// TIA Portal V16 export
// export: Created 2021-11-12T13:33:06.5426494Z, ExportSetting WithDefaults, DisplayName Totally Integrated Automation Portal, DisplayVersion V16 Update 3, DisplayName TIA Portal Version Control Interface, DisplayVersion V16 Update 2, DisplayName TIA Portal Openness, DisplayVersion V16 Update 3, DisplayName SINAMICS Startdrive Advanced, DisplayVersion V16 Update 5, DisplayName SINAMICS Startdrive G130, G150, S120, S150, SINAMICS MV, S210, DisplayVersion V16 Update 5, DisplayName SINAMICS Startdrive G110M, G120, G120C, G120D, G120P, G115D, DisplayVersion V16 Update 5, DisplayName STEP 7 Professional, DisplayVersion V16 Update 3, DisplayName STEP 7 Safety, DisplayVersion V16, DisplayName WinCC UA Professional, DisplayVersion V16 Update 3
FUNCTION_BLOCK "Station410"   // FB83, LAD
{ S7_Optimized_Access := 'TRUE' }
VERSION : 0.1
// stored: AutoNumber true, IsIECCheckEnabled false, IsRetainMemResEnabled false, MemoryReserve 100, SetENOAutomatically false, UDAEnableTagReadback false
   VAR
      "SF_EQ01-MA01" : "STD_Drive1";   // Water pump (P31)
      "SF_EQ01-MA02" : "STD_Valve2WB";   // Valve with servomotor (A1417)
      "SF_EQ01-MA03" : "STD_Valve2WB";   // Valve with servomotor (A1414)
      "SF_EQ01-MA04" : "STD_Valve2WB";   // Valve with servomotor (A1411)
      "SF_UC11-TA01" { S7_SetPoint := 'True'} : "STD_Siemens_G120_CU240E_2_PN";   // Conveyor
      SF_Alarm1 { S7_SetPoint := 'True'} : "STD_DI_Mon";   // Sensor Max level active and sensor Min level
      SF_Alarm2 { S7_SetPoint := 'True'} : "STD_DI_Mon";   // Sensor Min level active and analog level sensor under 10%
      SF_Alarm3 { S7_SetPoint := 'True'} : "STD_DI_Mon";   // Analog level sensor over 40% and sensor min level not active
      SF_Alarm4 { S7_SetPoint := 'True'} : "STD_DI_Mon";   // Water temperature high
      SF_Alarm5 { S7_SetPoint := 'True'} : "STD_DI_Mon";   // Water temperature low
      SF_Alarm6 { S7_SetPoint := 'True'} : "STD_DI_Mon";   // Water level high
      SF_Alarm7 { S7_SetPoint := 'True'} : "STD_DI_Mon";   // BSN 5 tacts and water level NOK
      SF_Alarm8 { S7_SetPoint := 'True'} : "STD_DI_Mon";   // Filling and no water level change
      SF_Alarm9 { S7_SetPoint := 'True'} : "STD_DI_Mon";   // Drain and no water level change
      SS_Cooling : Struct
         LiqTemp : Real;   // Real temperature of liquid
         HystMin : Real;   // Minimal hysteresis of requested temperature for cooling liquid
         HystMax : Real;   // Maximal hysteresis of requested temperature for cooling liquid
         RunPump : Bool;
         RegEn : Bool;   // Enable regulation
      END_STRUCT;
      SR_TmpWaterLevel : Real;
      SB1_PowerOk { S7_SetPoint := 'True'} : Bool;
      SF_TimerWaterHom { S7_SetPoint := 'True'} : TON_TIME;
   END_VAR
   VAR_TEMP
      TS_EQ01MA01 : "UDT_DriveControl";   // Water pump (P31)
      TS_EQ01MA02 : "UDT_DriveControl";   // Valve with servomotor (A1417)
      TS_EQ01MA03 : "UDT_DriveControl";   // Valve with servomotor (A1414)
      TS_EQ01MA04 : "UDT_DriveControl";   // Valve with servomotor (A1411)
      TS_UC11TA01 : Struct   // Conveyor
         ReqDir1 : Bool;   // Move in direction 1
         ReqDir2 : Bool;   // Move in direction 2
         AckErr : Bool;   // Acknowledge error
         SpeedSP : Real;   // Speed setpoint
      END_STRUCT;
      TS_CirculationValve : Struct
         HystMin : Real;
         HystMax : Real;
         SP : Real;
      END_STRUCT;
      TB1_WaterHom : Bool;   // Water homogenization is not done
   END_VAR
   VAR CONSTANT
      CI_EQ01MA03_hyst : SInt := 2;   // Valve hysteresis
   END_VAR
   VAR_TEMP   // added for the SCL form of the ladder/FBD networks
      _w1 : Bool;
   END_VAR
BEGIN

REGION Network 2: ***************ClearTemporary***************
END_REGION

REGION Network 3: ***************SesorsAlarms***************
END_REGION

REGION Network 4: Alarm - Sensor Max level active and sensor Min level Not Active
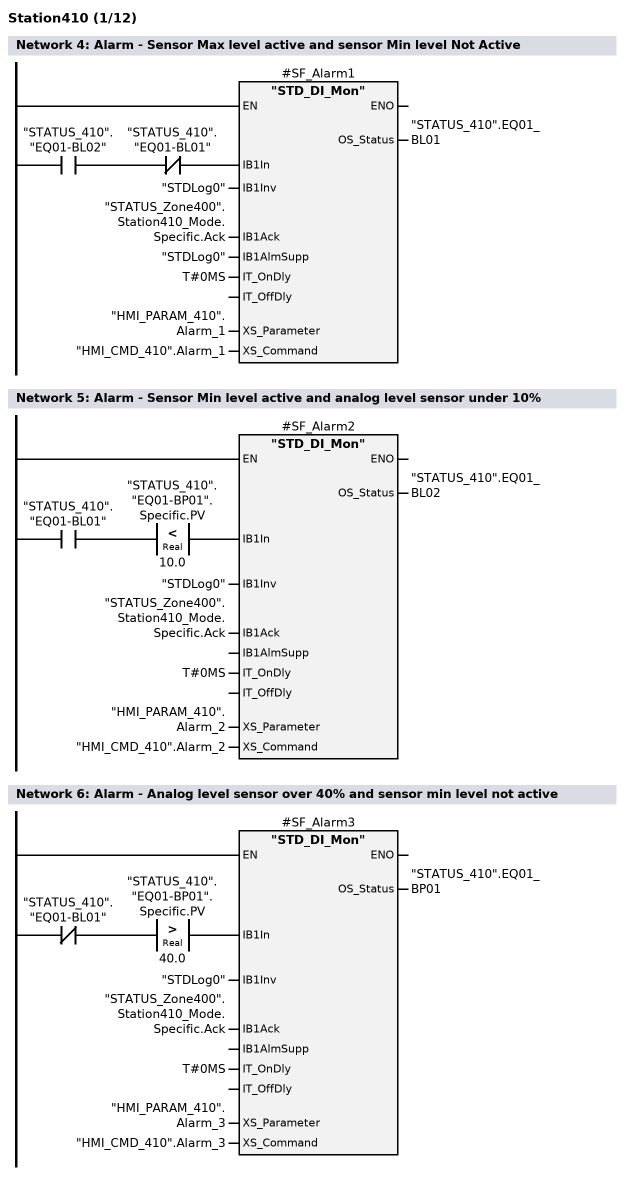
   RUNG wire#powerrail
      #SF_Alarm1(IB1In := wire#w1, IB1Inv := "STDLog0", IB1Ack := "STATUS_Zone400".Station410_Mode.Specific.Ack, IB1AlmSupp := "STDLog0", IT_OnDly := T#0MS, IT_OffDly :=, XS_Parameter := "HMI_PARAM_410".Alarm_1, XS_Command := "HMI_CMD_410".Alarm_1, OS_Status => "STATUS_410".EQ01_BL01)
   END_RUNG
   RUNG wire#powerrail
      Contact( "STATUS_410"."EQ01-BL02" )
      I_Contact( "STATUS_410"."EQ01-BL01" )
   END_RUNG wire#w1
   // the same network as SCL:
   #SF_Alarm1(IB1In := "STATUS_410"."EQ01-BL02" AND NOT "STATUS_410"."EQ01-BL01",   // "STD_DI_Mon"
              IB1Inv := "STDLog0",
              IB1Ack := "STATUS_Zone400".Station410_Mode.Specific.Ack,
              IB1AlmSupp := "STDLog0",
              IT_OnDly := T#0MS,
              XS_Parameter := "HMI_PARAM_410".Alarm_1,
              XS_Command := "HMI_CMD_410".Alarm_1,
              OS_Status => "STATUS_410".EQ01_BL01);
END_REGION

REGION Network 5: Alarm - Sensor Min level active and analog level sensor under 10%
   RUNG wire#powerrail
      #SF_Alarm2(IB1In := wire#w1, IB1Inv := "STDLog0", IB1Ack := "STATUS_Zone400".Station410_Mode.Specific.Ack, IB1AlmSupp :=, IT_OnDly := T#0MS, IT_OffDly :=, XS_Parameter := "HMI_PARAM_410".Alarm_2, XS_Command := "HMI_CMD_410".Alarm_2, OS_Status => "STATUS_410".EQ01_BL02)
   END_RUNG
   RUNG wire#powerrail
      Contact( "STATUS_410"."EQ01-BL01" )
      { S7_Templates := "SrcType := Real" } LT_Contact(in1 := "STATUS_410"."EQ01-BP01".Specific.PV, in2 := 10.0)
   END_RUNG wire#w1
   // the same network as SCL:
   #SF_Alarm2(IB1In := "STATUS_410"."EQ01-BL01" AND ("STATUS_410"."EQ01-BP01".Specific.PV < 10.0),   // "STD_DI_Mon"
              IB1Inv := "STDLog0",
              IB1Ack := "STATUS_Zone400".Station410_Mode.Specific.Ack,
              IT_OnDly := T#0MS,
              XS_Parameter := "HMI_PARAM_410".Alarm_2,
              XS_Command := "HMI_CMD_410".Alarm_2,
              OS_Status => "STATUS_410".EQ01_BL02);
END_REGION

REGION Network 6: Alarm - Analog level sensor over 40% and sensor min level not active
   RUNG wire#powerrail
      #SF_Alarm3(IB1In := wire#w1, IB1Inv := "STDLog0", IB1Ack := "STATUS_Zone400".Station410_Mode.Specific.Ack, IB1AlmSupp :=, IT_OnDly := T#0MS, IT_OffDly :=, XS_Parameter := "HMI_PARAM_410".Alarm_3, XS_Command := "HMI_CMD_410".Alarm_3, OS_Status => "STATUS_410".EQ01_BP01)
   END_RUNG
   RUNG wire#powerrail
      I_Contact( "STATUS_410"."EQ01-BL01" )
      { S7_Templates := "SrcType := Real" } GT_Contact(in1 := "STATUS_410"."EQ01-BP01".Specific.PV, in2 := 40.0)
   END_RUNG wire#w1
   // the same network as SCL:
   #SF_Alarm3(IB1In := NOT "STATUS_410"."EQ01-BL01" AND ("STATUS_410"."EQ01-BP01".Specific.PV > 40.0),   // "STD_DI_Mon"
              IB1Inv := "STDLog0",
              IB1Ack := "STATUS_Zone400".Station410_Mode.Specific.Ack,
              IT_OnDly := T#0MS,
              XS_Parameter := "HMI_PARAM_410".Alarm_3,
              XS_Command := "HMI_CMD_410".Alarm_3,
              OS_Status => "STATUS_410".EQ01_BP01);
END_REGION

REGION Network 7: ***************ProcesAlarms***************
END_REGION

REGION Network 8: Alarm - Water temperature high
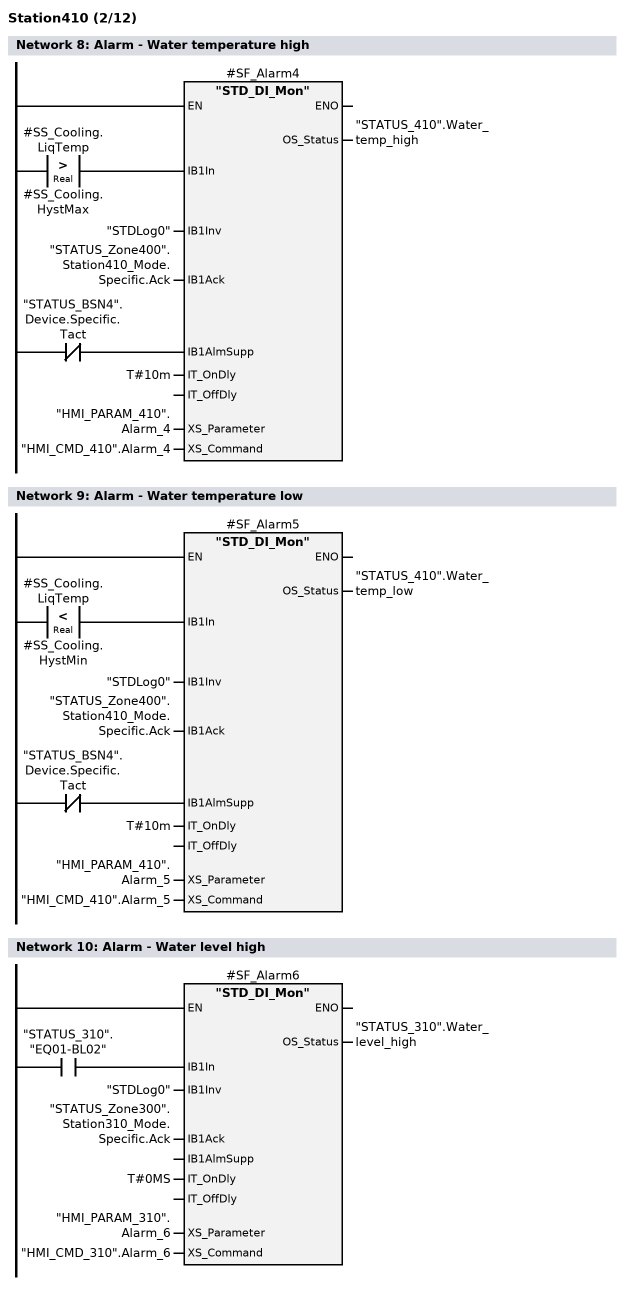
   RUNG wire#powerrail
      #SF_Alarm4(IB1In := wire#w1, IB1AlmSupp := wire#w2, IB1Inv := "STDLog0", IB1Ack := "STATUS_Zone400".Station410_Mode.Specific.Ack, IT_OnDly := T#10m, IT_OffDly :=, XS_Parameter := "HMI_PARAM_410".Alarm_4, XS_Command := "HMI_CMD_410".Alarm_4, OS_Status => "STATUS_410".Water_temp_high)
   END_RUNG
   RUNG wire#powerrail
      { S7_Templates := "SrcType := Real" } GT_Contact(in1 := #SS_Cooling.LiqTemp, in2 := #SS_Cooling.HystMax)
   END_RUNG wire#w1
   RUNG wire#powerrail
      I_Contact( "STATUS_BSN4".Device.Specific.Tact )
   END_RUNG wire#w2
   // the same network as SCL:
   #SF_Alarm4(IB1In := #SS_Cooling.LiqTemp > #SS_Cooling.HystMax,   // "STD_DI_Mon"
              IB1Inv := "STDLog0",
              IB1Ack := "STATUS_Zone400".Station410_Mode.Specific.Ack,
              IB1AlmSupp := NOT "STATUS_BSN4".Device.Specific.Tact,
              IT_OnDly := T#10m,
              XS_Parameter := "HMI_PARAM_410".Alarm_4,
              XS_Command := "HMI_CMD_410".Alarm_4,
              OS_Status => "STATUS_410".Water_temp_high);
END_REGION

REGION Network 9: Alarm - Water temperature low
   RUNG wire#powerrail
      #SF_Alarm5(IB1In := wire#w1, IB1AlmSupp := wire#w2, IB1Inv := "STDLog0", IB1Ack := "STATUS_Zone400".Station410_Mode.Specific.Ack, IT_OnDly := T#10m, IT_OffDly :=, XS_Parameter := "HMI_PARAM_410".Alarm_5, XS_Command := "HMI_CMD_410".Alarm_5, OS_Status => "STATUS_410".Water_temp_low)
   END_RUNG
   RUNG wire#powerrail
      { S7_Templates := "SrcType := Real" } LT_Contact(in1 := #SS_Cooling.LiqTemp, in2 := #SS_Cooling.HystMin)
   END_RUNG wire#w1
   RUNG wire#powerrail
      I_Contact( "STATUS_BSN4".Device.Specific.Tact )
   END_RUNG wire#w2
   // the same network as SCL:
   #SF_Alarm5(IB1In := #SS_Cooling.LiqTemp < #SS_Cooling.HystMin,   // "STD_DI_Mon"
              IB1Inv := "STDLog0",
              IB1Ack := "STATUS_Zone400".Station410_Mode.Specific.Ack,
              IB1AlmSupp := NOT "STATUS_BSN4".Device.Specific.Tact,
              IT_OnDly := T#10m,
              XS_Parameter := "HMI_PARAM_410".Alarm_5,
              XS_Command := "HMI_CMD_410".Alarm_5,
              OS_Status => "STATUS_410".Water_temp_low);
END_REGION

REGION Network 10: Alarm - Water level high
   RUNG wire#powerrail
      #SF_Alarm6(IB1In := wire#w1, IB1Inv := "STDLog0", IB1Ack := "STATUS_Zone300".Station310_Mode.Specific.Ack, IB1AlmSupp :=, IT_OnDly := T#0MS, IT_OffDly :=, XS_Parameter := "HMI_PARAM_310".Alarm_6, XS_Command := "HMI_CMD_310".Alarm_6, OS_Status => "STATUS_310".Water_level_high)
   END_RUNG
   RUNG wire#powerrail
      Contact( "STATUS_310"."EQ01-BL02" )
   END_RUNG wire#w1
   // the same network as SCL:
   #SF_Alarm6(IB1In := "STATUS_310"."EQ01-BL02",   // "STD_DI_Mon"
              IB1Inv := "STDLog0",
              IB1Ack := "STATUS_Zone300".Station310_Mode.Specific.Ack,
              IT_OnDly := T#0MS,
              XS_Parameter := "HMI_PARAM_310".Alarm_6,
              XS_Command := "HMI_CMD_310".Alarm_6,
              OS_Status => "STATUS_310".Water_level_high);
END_REGION

REGION Network 11: Alarm - BSN5 tacts and water level NOK
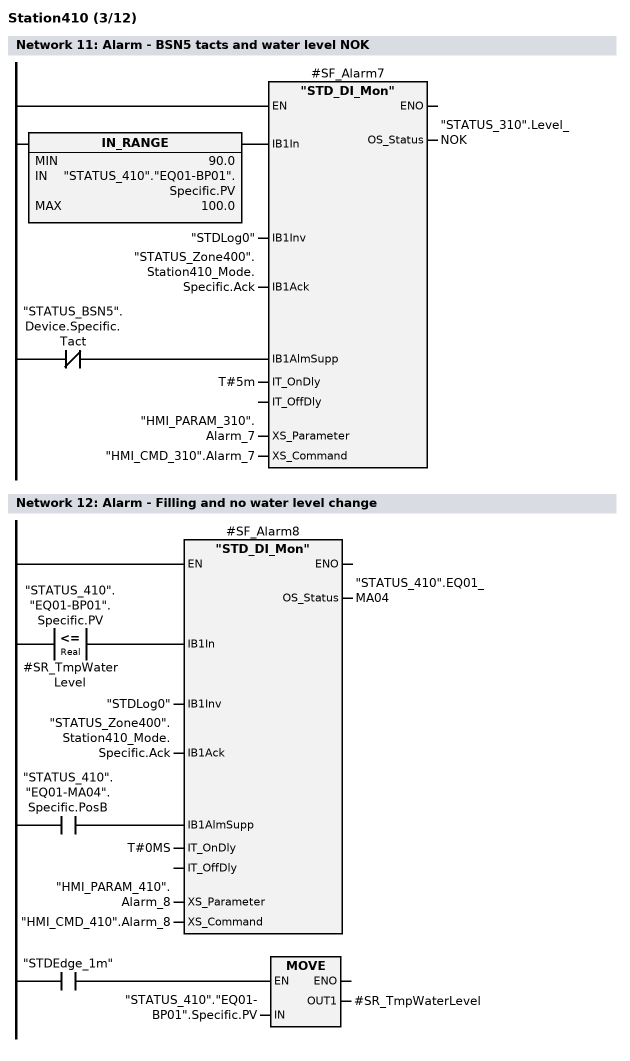
   RUNG wire#powerrail
      #SF_Alarm7(IB1In := wire#w1, IB1AlmSupp := wire#w2, IB1Inv := "STDLog0", IB1Ack := "STATUS_Zone400".Station410_Mode.Specific.Ack, IT_OnDly := T#5m, IT_OffDly :=, XS_Parameter := "HMI_PARAM_310".Alarm_7, XS_Command := "HMI_CMD_310".Alarm_7, OS_Status => "STATUS_310".Level_NOK)
   END_RUNG
   RUNG wire#powerrail
      { S7_Templates := "SrcType := Real" } InRange(min := 90.0, in := "STATUS_410"."EQ01-BP01".Specific.PV, max := 100.0)
   END_RUNG wire#w1
   RUNG wire#powerrail
      I_Contact( "STATUS_BSN5".Device.Specific.Tact )
   END_RUNG wire#w2
   // the same network as SCL:
   #SF_Alarm7(IB1In := (90.0 <= "STATUS_410"."EQ01-BP01".Specific.PV) AND ("STATUS_410"."EQ01-BP01".Specific.PV <= 100.0),   // "STD_DI_Mon"
              IB1Inv := "STDLog0",
              IB1Ack := "STATUS_Zone400".Station410_Mode.Specific.Ack,
              IB1AlmSupp := NOT "STATUS_BSN5".Device.Specific.Tact,
              IT_OnDly := T#5m,
              XS_Parameter := "HMI_PARAM_310".Alarm_7,
              XS_Command := "HMI_CMD_310".Alarm_7,
              OS_Status => "STATUS_310".Level_NOK);
END_REGION

REGION Network 12: Alarm - Filling and no water level change
   RUNG wire#powerrail
      #SF_Alarm8(IB1In := wire#w1, IB1AlmSupp := wire#w2, IB1Inv := "STDLog0", IB1Ack := "STATUS_Zone400".Station410_Mode.Specific.Ack, IT_OnDly := T#0MS, IT_OffDly :=, XS_Parameter := "HMI_PARAM_410".Alarm_8, XS_Command := "HMI_CMD_410".Alarm_8, OS_Status => "STATUS_410".EQ01_MA04)
   END_RUNG
   RUNG wire#powerrail
      { S7_Templates := "SrcType := Real" } LE_Contact(in1 := "STATUS_410"."EQ01-BP01".Specific.PV, in2 := #SR_TmpWaterLevel)
   END_RUNG wire#w1
   RUNG wire#powerrail
      Contact( "STATUS_410"."EQ01-MA04".Specific.PosB )
   END_RUNG wire#w2
   RUNG wire#powerrail
      Contact( "STDEdge_1m" )
      Move(in := "STATUS_410"."EQ01-BP01".Specific.PV, out1 => #SR_TmpWaterLevel)
   END_RUNG
   // the same network as SCL:
   #SF_Alarm8(IB1In := "STATUS_410"."EQ01-BP01".Specific.PV <= #SR_TmpWaterLevel,   // "STD_DI_Mon"
              IB1Inv := "STDLog0",
              IB1Ack := "STATUS_Zone400".Station410_Mode.Specific.Ack,
              IB1AlmSupp := "STATUS_410"."EQ01-MA04".Specific.PosB,
              IT_OnDly := T#0MS,
              XS_Parameter := "HMI_PARAM_410".Alarm_8,
              XS_Command := "HMI_CMD_410".Alarm_8,
              OS_Status => "STATUS_410".EQ01_MA04);
   IF "STDEdge_1m" THEN #SR_TmpWaterLevel := "STATUS_410"."EQ01-BP01".Specific.PV; END_IF;
END_REGION

REGION Network 13: Alarm - Drain and no water level change
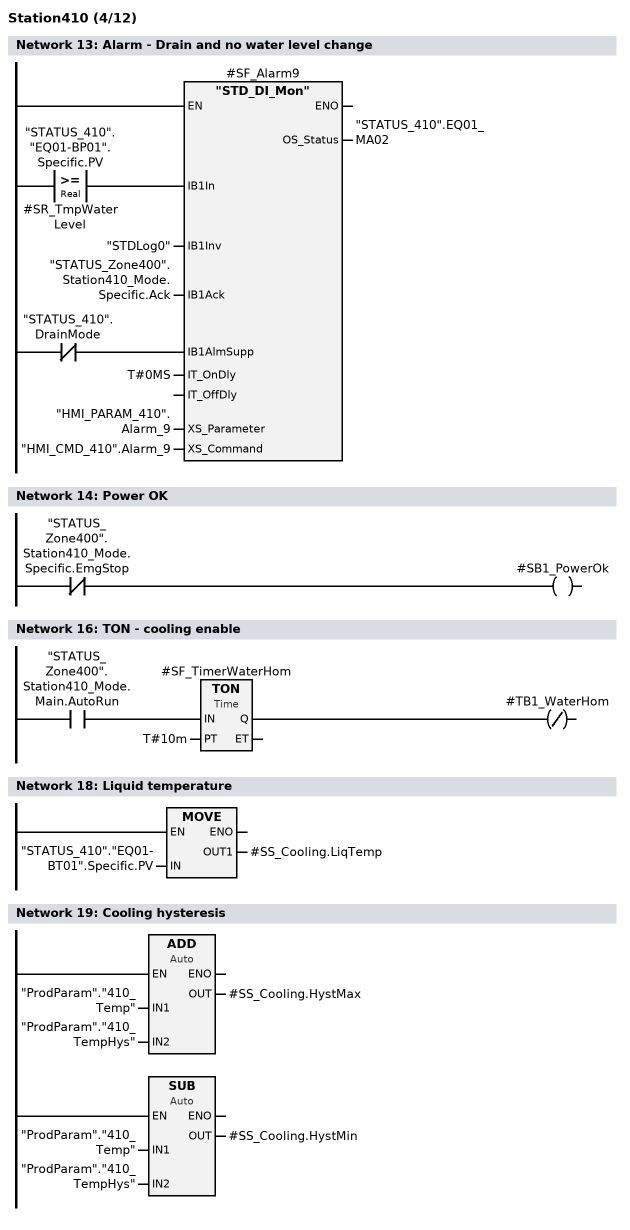
   RUNG wire#powerrail
      #SF_Alarm9(IB1In := wire#w1, IB1AlmSupp := wire#w2, IB1Inv := "STDLog0", IB1Ack := "STATUS_Zone400".Station410_Mode.Specific.Ack, IT_OnDly := T#0MS, IT_OffDly :=, XS_Parameter := "HMI_PARAM_410".Alarm_9, XS_Command := "HMI_CMD_410".Alarm_9, OS_Status => "STATUS_410".EQ01_MA02)
   END_RUNG
   RUNG wire#powerrail
      { S7_Templates := "SrcType := Real" } GE_Contact(in1 := "STATUS_410"."EQ01-BP01".Specific.PV, in2 := #SR_TmpWaterLevel)
   END_RUNG wire#w1
   RUNG wire#powerrail
      I_Contact( "STATUS_410".DrainMode )
   END_RUNG wire#w2
   // the same network as SCL:
   #SF_Alarm9(IB1In := "STATUS_410"."EQ01-BP01".Specific.PV >= #SR_TmpWaterLevel,   // "STD_DI_Mon"
              IB1Inv := "STDLog0",
              IB1Ack := "STATUS_Zone400".Station410_Mode.Specific.Ack,
              IB1AlmSupp := NOT "STATUS_410".DrainMode,
              IT_OnDly := T#0MS,
              XS_Parameter := "HMI_PARAM_410".Alarm_9,
              XS_Command := "HMI_CMD_410".Alarm_9,
              OS_Status => "STATUS_410".EQ01_MA02);
END_REGION

REGION Network 14: Power OK
   RUNG wire#powerrail
      I_Contact( "STATUS_Zone400".Station410_Mode.Specific.EmgStop )
      Coil( #SB1_PowerOk )
   END_RUNG
   // the same network as SCL:
   #SB1_PowerOk := NOT "STATUS_Zone400".Station410_Mode.Specific.EmgStop;
END_REGION

REGION Network 15: ********** Water homogenization **********
END_REGION

REGION Network 16: TON - cooling enable
   RUNG wire#powerrail
      Contact( "STATUS_Zone400".Station410_Mode.Main.AutoRun )
      { S7_Templates := "time_type := Time" } #SF_TimerWaterHom.TON(pt := T#10m, et =>)
      I_Coil( #TB1_WaterHom )
   END_RUNG
   // the same network as SCL:
   #SF_TimerWaterHom(IN := "STATUS_Zone400".Station410_Mode.Main.AutoRun, PT := T#10m);   // TON
   #TB1_WaterHom := NOT #SF_TimerWaterHom.Q;
END_REGION

REGION Network 17: ********** Cooling **********
END_REGION

REGION Network 18: Liquid temperature
   RUNG wire#powerrail
      Move(in := "STATUS_410"."EQ01-BT01".Specific.PV, out1 => #SS_Cooling.LiqTemp)
   END_RUNG
   // the same network as SCL:
   #SS_Cooling.LiqTemp := "STATUS_410"."EQ01-BT01".Specific.PV;
END_REGION

REGION Network 19: Cooling hysteresis
   RUNG wire#powerrail
      Add(in1 := "ProdParam"."410_Temp", in2 := "ProdParam"."410_TempHys", out => #SS_Cooling.HystMax)
   END_RUNG
   RUNG wire#powerrail
      Sub(in1 := "ProdParam"."410_Temp", in2 := "ProdParam"."410_TempHys", out => #SS_Cooling.HystMin)
   END_RUNG
   // the same network as SCL:
   #SS_Cooling.HystMax := "ProdParam"."410_Temp" + "ProdParam"."410_TempHys";
   #SS_Cooling.HystMin := "ProdParam"."410_Temp" - "ProdParam"."410_TempHys";
END_REGION

REGION Network 20: EQ01-MA03 regulation enable
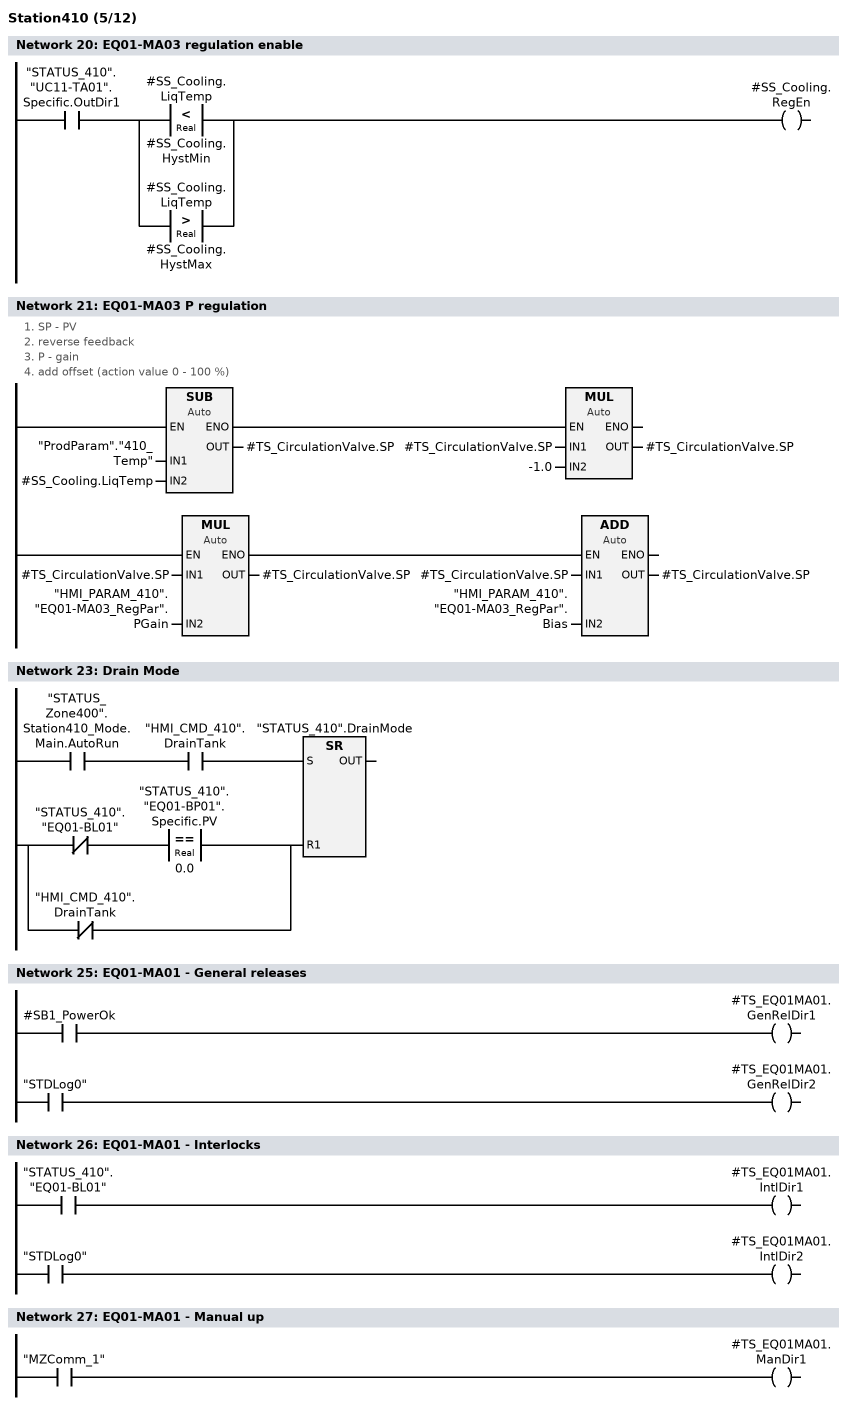
   RUNG wire#powerrail
      Contact( "STATUS_410"."UC11-TA01".Specific.OutDir1 )
      wire#w1
      { S7_Templates := "SrcType := Real" } LT_Contact(in1 := #SS_Cooling.LiqTemp, in2 := #SS_Cooling.HystMin)
      wire#w2
      Coil( #SS_Cooling.RegEn )
   END_RUNG
   RUNG wire#w1
      { S7_Templates := "SrcType := Real" } GT_Contact(in1 := #SS_Cooling.LiqTemp, in2 := #SS_Cooling.HystMax)
   END_RUNG wire#w2
   // the same network as SCL:
   #SS_Cooling.RegEn := "STATUS_410"."UC11-TA01".Specific.OutDir1 AND ((#SS_Cooling.LiqTemp < #SS_Cooling.HystMin) OR (#SS_Cooling.LiqTemp > #SS_Cooling.HystMax));
END_REGION

REGION Network 21: EQ01-MA03 P regulation
   // 1. SP - PV
   // 2. reverse feedback
   // 3. P - gain
   // 4. add offset (action value 0 - 100 %)
   RUNG wire#powerrail
      Sub(in1 := "ProdParam"."410_Temp", in2 := #SS_Cooling.LiqTemp, out => #TS_CirculationValve.SP)
      Mul(in1 := #TS_CirculationValve.SP, in2 := -1.0, out => #TS_CirculationValve.SP)
   END_RUNG
   RUNG wire#powerrail
      Mul(in1 := #TS_CirculationValve.SP, in2 := "HMI_PARAM_410"."EQ01-MA03_RegPar".PGain, out => #TS_CirculationValve.SP)
      Add(in1 := #TS_CirculationValve.SP, in2 := "HMI_PARAM_410"."EQ01-MA03_RegPar".Bias, out => #TS_CirculationValve.SP)
   END_RUNG
   // the same network as SCL:
   #TS_CirculationValve.SP := "ProdParam"."410_Temp" - #SS_Cooling.LiqTemp;
   #TS_CirculationValve.SP := #TS_CirculationValve.SP * (-1.0);
   #TS_CirculationValve.SP := #TS_CirculationValve.SP * "HMI_PARAM_410"."EQ01-MA03_RegPar".PGain;
   #TS_CirculationValve.SP := #TS_CirculationValve.SP + "HMI_PARAM_410"."EQ01-MA03_RegPar".Bias;
END_REGION

REGION Network 22: ********** Draining **********
END_REGION

REGION Network 23: Drain Mode
   RUNG wire#powerrail
      Contact( "STATUS_Zone400".Station410_Mode.Main.AutoRun )
      Contact( "HMI_CMD_410".DrainTank )
      S_SR(operand := "STATUS_410".DrainMode, r1 := wire#w1)
   END_RUNG
   RUNG wire#powerrail
      I_Contact( "STATUS_410"."EQ01-BL01" )
      { S7_Templates := "SrcType := Real" } EQ_Contact(in1 := "STATUS_410"."EQ01-BP01".Specific.PV, in2 := 0.0)
   END_RUNG wire#w1
   RUNG wire#powerrail
      I_Contact( "HMI_CMD_410".DrainTank )
   END_RUNG wire#w1
   // the same network as SCL:
   IF "STATUS_Zone400".Station410_Mode.Main.AutoRun AND "HMI_CMD_410".DrainTank THEN
       "STATUS_410".DrainMode := TRUE;   // SR flip-flop
   END_IF;
   IF (NOT "STATUS_410"."EQ01-BL01" AND ("STATUS_410"."EQ01-BP01".Specific.PV = 0.0)) OR NOT "HMI_CMD_410".DrainTank THEN
       "STATUS_410".DrainMode := FALSE;
   END_IF;
END_REGION

REGION Network 24: ********** Circulation Pump EQ01-MA01 **********
END_REGION

REGION Network 25: EQ01-MA01 - General releases
   RUNG wire#powerrail
      Contact( #SB1_PowerOk )
      Coil( #TS_EQ01MA01.GenRelDir1 )
   END_RUNG
   RUNG wire#powerrail
      Contact( "STDLog0" )
      Coil( #TS_EQ01MA01.GenRelDir2 )
   END_RUNG
   // the same network as SCL:
   #TS_EQ01MA01.GenRelDir1 := #SB1_PowerOk;
   #TS_EQ01MA01.GenRelDir2 := "STDLog0";
END_REGION

REGION Network 26: EQ01-MA01 - Interlocks
   RUNG wire#powerrail
      Contact( "STATUS_410"."EQ01-BL01" )
      Coil( #TS_EQ01MA01.IntlDir1 )
   END_RUNG
   RUNG wire#powerrail
      Contact( "STDLog0" )
      Coil( #TS_EQ01MA01.IntlDir2 )
   END_RUNG
   // the same network as SCL:
   #TS_EQ01MA01.IntlDir1 := "STATUS_410"."EQ01-BL01";
   #TS_EQ01MA01.IntlDir2 := "STDLog0";
END_REGION

REGION Network 27: EQ01-MA01 - Manual up
   RUNG wire#powerrail
      Contact( "MZComm_1" )
      Coil( #TS_EQ01MA01.ManDir1 )
   END_RUNG
   // the same network as SCL:
   #TS_EQ01MA01.ManDir1 := "MZComm_1";
END_REGION

REGION Network 28: EQ01-MA01 - Manual down
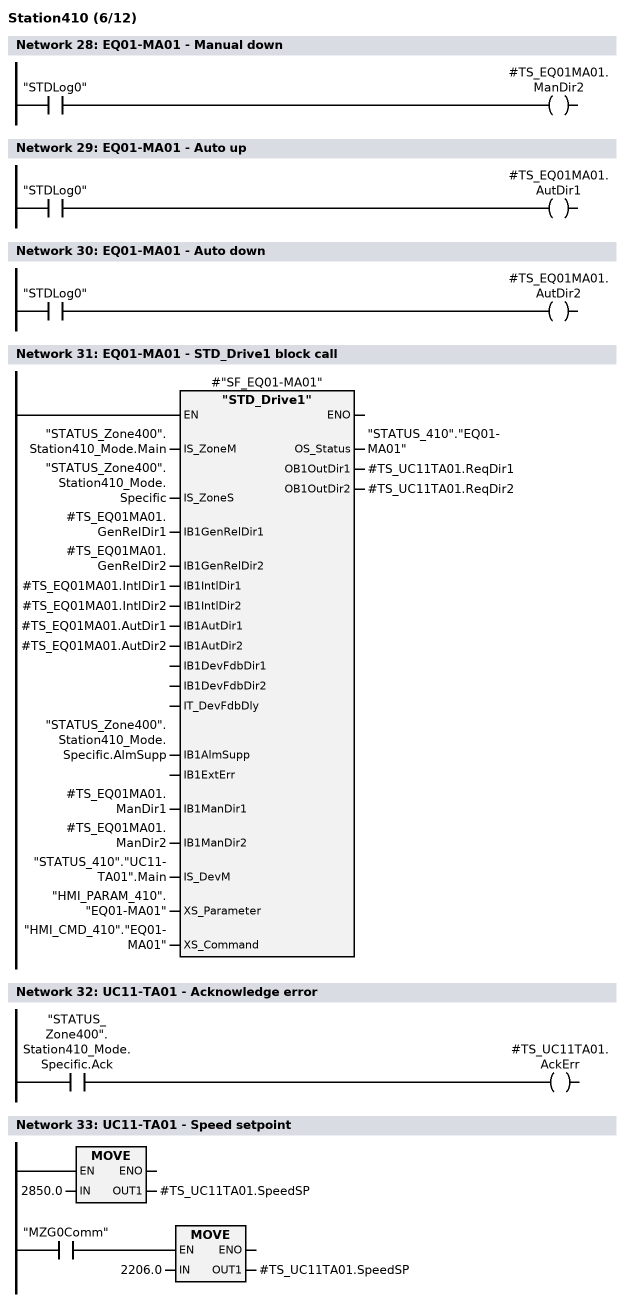
   RUNG wire#powerrail
      Contact( "STDLog0" )
      Coil( #TS_EQ01MA01.ManDir2 )
   END_RUNG
   // the same network as SCL:
   #TS_EQ01MA01.ManDir2 := "STDLog0";
END_REGION

REGION Network 29: EQ01-MA01 - Auto up
   RUNG wire#powerrail
      Contact( "STDLog0" )
      Coil( #TS_EQ01MA01.AutDir1 )
   END_RUNG
   // the same network as SCL:
   #TS_EQ01MA01.AutDir1 := "STDLog0";
END_REGION

REGION Network 30: EQ01-MA01 - Auto down
   RUNG wire#powerrail
      Contact( "STDLog0" )
      Coil( #TS_EQ01MA01.AutDir2 )
   END_RUNG
   // the same network as SCL:
   #TS_EQ01MA01.AutDir2 := "STDLog0";
END_REGION

REGION Network 31: EQ01-MA01 - STD_Drive1 block call
   RUNG wire#powerrail
      #"SF_EQ01-MA01"(IS_ZoneM := "STATUS_Zone400".Station410_Mode.Main, IS_ZoneS := "STATUS_Zone400".Station410_Mode.Specific, IB1GenRelDir1 := #TS_EQ01MA01.GenRelDir1, IB1GenRelDir2 := #TS_EQ01MA01.GenRelDir2, IB1IntlDir1 := #TS_EQ01MA01.IntlDir1, IB1IntlDir2 := #TS_EQ01MA01.IntlDir2, IB1AutDir1 := #TS_EQ01MA01.AutDir1, IB1AutDir2 := #TS_EQ01MA01.AutDir2, IB1DevFdbDir1 :=, IB1DevFdbDir2 :=, IT_DevFdbDly :=, IB1AlmSupp := "STATUS_Zone400".Station410_Mode.Specific.AlmSupp, IB1ExtErr :=, IB1ManDir1 := #TS_EQ01MA01.ManDir1, IB1ManDir2 := #TS_EQ01MA01.ManDir2, IS_DevM := "STATUS_410"."UC11-TA01".Main, XS_Parameter := "HMI_PARAM_410"."EQ01-MA01", XS_Command := "HMI_CMD_410"."EQ01-MA01", OS_Status => "STATUS_410"."EQ01-MA01", OB1OutDir1 => #TS_UC11TA01.ReqDir1, OB1OutDir2 => #TS_UC11TA01.ReqDir2)
   END_RUNG
   // the same network as SCL:
   #"SF_EQ01-MA01"(IS_ZoneM := "STATUS_Zone400".Station410_Mode.Main,   // "STD_Drive1"
                   IS_ZoneS := "STATUS_Zone400".Station410_Mode.Specific,
                   IB1GenRelDir1 := #TS_EQ01MA01.GenRelDir1,
                   IB1GenRelDir2 := #TS_EQ01MA01.GenRelDir2,
                   IB1IntlDir1 := #TS_EQ01MA01.IntlDir1,
                   IB1IntlDir2 := #TS_EQ01MA01.IntlDir2,
                   IB1AutDir1 := #TS_EQ01MA01.AutDir1,
                   IB1AutDir2 := #TS_EQ01MA01.AutDir2,
                   IB1AlmSupp := "STATUS_Zone400".Station410_Mode.Specific.AlmSupp,
                   IB1ManDir1 := #TS_EQ01MA01.ManDir1,
                   IB1ManDir2 := #TS_EQ01MA01.ManDir2,
                   IS_DevM := "STATUS_410"."UC11-TA01".Main,
                   XS_Parameter := "HMI_PARAM_410"."EQ01-MA01",
                   XS_Command := "HMI_CMD_410"."EQ01-MA01",
                   OS_Status => "STATUS_410"."EQ01-MA01",
                   OB1OutDir1 => #TS_UC11TA01.ReqDir1,
                   OB1OutDir2 => #TS_UC11TA01.ReqDir2);
END_REGION

REGION Network 32: UC11-TA01 - Acknowledge error
   RUNG wire#powerrail
      Contact( "STATUS_Zone400".Station410_Mode.Specific.Ack )
      Coil( #TS_UC11TA01.AckErr )
   END_RUNG
   // the same network as SCL:
   #TS_UC11TA01.AckErr := "STATUS_Zone400".Station410_Mode.Specific.Ack;
END_REGION

REGION Network 33: UC11-TA01 - Speed setpoint
   RUNG wire#powerrail
      Move(in := 2850.0, out1 => #TS_UC11TA01.SpeedSP)
   END_RUNG
   RUNG wire#powerrail
      Contact( "MZG0Comm" )
      Move(in := 2206.0, out1 => #TS_UC11TA01.SpeedSP)
   END_RUNG
   // the same network as SCL:
   #TS_UC11TA01.SpeedSP := 2850.0;
   IF "MZG0Comm" THEN #TS_UC11TA01.SpeedSP := 2206.0; END_IF;
END_REGION

REGION Network 34: UC11-TA01 - Sinamics G120 STD block call (frequency convertor)
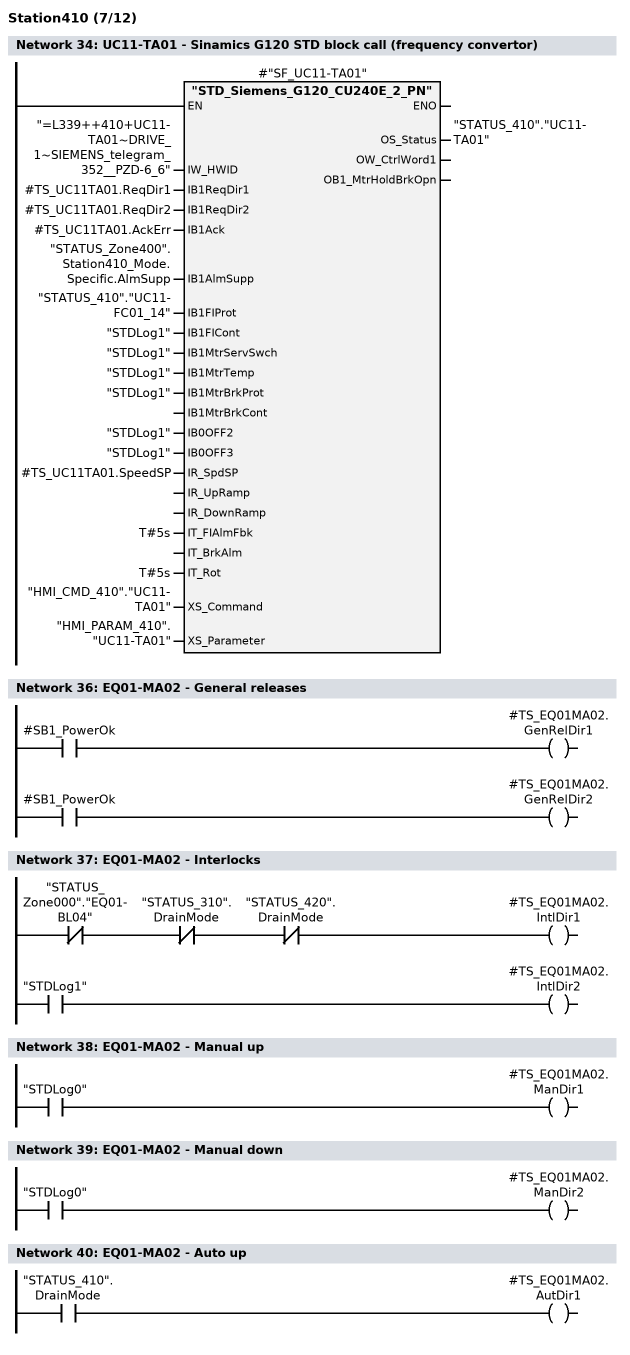
   RUNG wire#powerrail
      #"SF_UC11-TA01"(IW_HWID := "=L339++410+UC11-TA01~DRIVE_1~SIEMENS_telegram_352__PZD-6_6", IB1ReqDir1 := #TS_UC11TA01.ReqDir1, IB1ReqDir2 := #TS_UC11TA01.ReqDir2, IB1Ack := #TS_UC11TA01.AckErr, IB1AlmSupp := "STATUS_Zone400".Station410_Mode.Specific.AlmSupp, IB1FIProt := "STATUS_410"."UC11-FC01_14", IB1FICont := "STDLog1", IB1MtrServSwch := "STDLog1", IB1MtrTemp := "STDLog1", IB1MtrBrkProt := "STDLog1", IB1MtrBrkCont :=, IB0OFF2 := "STDLog1", IB0OFF3 := "STDLog1", IR_SpdSP := #TS_UC11TA01.SpeedSP, IR_UpRamp :=, IR_DownRamp :=, IT_FIAlmFbk := T#5s, IT_BrkAlm :=, IT_Rot := T#5s, XS_Command := "HMI_CMD_410"."UC11-TA01", XS_Parameter := "HMI_PARAM_410"."UC11-TA01", OS_Status => "STATUS_410"."UC11-TA01", OW_CtrlWord1 =>, OB1_MtrHoldBrkOpn =>)
   END_RUNG
   // the same network as SCL:
   #"SF_UC11-TA01"(IW_HWID := "=L339++410+UC11-TA01~DRIVE_1~SIEMENS_telegram_352__PZD-6_6",   // "STD_Siemens_G120_CU240E_2_PN"
                   IB1ReqDir1 := #TS_UC11TA01.ReqDir1,
                   IB1ReqDir2 := #TS_UC11TA01.ReqDir2,
                   IB1Ack := #TS_UC11TA01.AckErr,
                   IB1AlmSupp := "STATUS_Zone400".Station410_Mode.Specific.AlmSupp,
                   IB1FIProt := "STATUS_410"."UC11-FC01_14",
                   IB1FICont := "STDLog1",
                   IB1MtrServSwch := "STDLog1",
                   IB1MtrTemp := "STDLog1",
                   IB1MtrBrkProt := "STDLog1",
                   IB0OFF2 := "STDLog1",
                   IB0OFF3 := "STDLog1",
                   IR_SpdSP := #TS_UC11TA01.SpeedSP,
                   IT_FIAlmFbk := T#5s,
                   IT_Rot := T#5s,
                   XS_Command := "HMI_CMD_410"."UC11-TA01",
                   XS_Parameter := "HMI_PARAM_410"."UC11-TA01",
                   OS_Status => "STATUS_410"."UC11-TA01");
END_REGION

REGION Network 35: ********** Draining Valve EQ01-MA02 **********
END_REGION

REGION Network 36: EQ01-MA02 - General releases
   RUNG wire#powerrail
      Contact( #SB1_PowerOk )
      Coil( #TS_EQ01MA02.GenRelDir1 )
   END_RUNG
   RUNG wire#powerrail
      Contact( #SB1_PowerOk )
      Coil( #TS_EQ01MA02.GenRelDir2 )
   END_RUNG
   // the same network as SCL:
   #TS_EQ01MA02.GenRelDir1 := #SB1_PowerOk;
   #TS_EQ01MA02.GenRelDir2 := #SB1_PowerOk;
END_REGION

REGION Network 37: EQ01-MA02 - Interlocks
   RUNG wire#powerrail
      I_Contact( "STATUS_Zone000"."EQ01-BL04" )
      I_Contact( "STATUS_310".DrainMode )
      I_Contact( "STATUS_420".DrainMode )
      Coil( #TS_EQ01MA02.IntlDir1 )
   END_RUNG
   RUNG wire#powerrail
      Contact( "STDLog1" )
      Coil( #TS_EQ01MA02.IntlDir2 )
   END_RUNG
   // the same network as SCL:
   #TS_EQ01MA02.IntlDir1 := NOT "STATUS_Zone000"."EQ01-BL04" AND NOT "STATUS_310".DrainMode AND NOT "STATUS_420".DrainMode;
   #TS_EQ01MA02.IntlDir2 := "STDLog1";
END_REGION

REGION Network 38: EQ01-MA02 - Manual up
   RUNG wire#powerrail
      Contact( "STDLog0" )
      Coil( #TS_EQ01MA02.ManDir1 )
   END_RUNG
   // the same network as SCL:
   #TS_EQ01MA02.ManDir1 := "STDLog0";
END_REGION

REGION Network 39: EQ01-MA02 - Manual down
   RUNG wire#powerrail
      Contact( "STDLog0" )
      Coil( #TS_EQ01MA02.ManDir2 )
   END_RUNG
   // the same network as SCL:
   #TS_EQ01MA02.ManDir2 := "STDLog0";
END_REGION

REGION Network 40: EQ01-MA02 - Auto up
   RUNG wire#powerrail
      Contact( "STATUS_410".DrainMode )
      Coil( #TS_EQ01MA02.AutDir1 )
   END_RUNG
   // the same network as SCL:
   #TS_EQ01MA02.AutDir1 := "STATUS_410".DrainMode;
END_REGION

REGION Network 41: EQ01-MA02 - Auto down
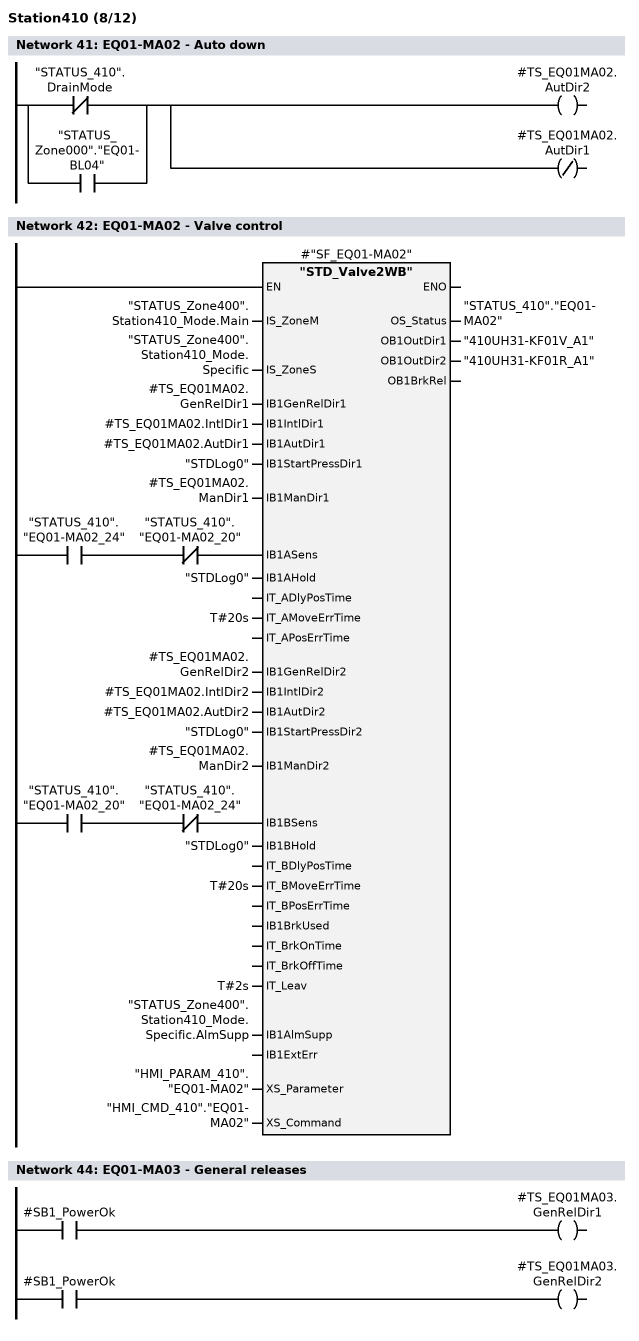
   RUNG wire#powerrail
      I_Contact( "STATUS_410".DrainMode )
      wire#w1
      Coil( #TS_EQ01MA02.AutDir2 )
   END_RUNG
   RUNG wire#powerrail
      Contact( "STATUS_Zone000"."EQ01-BL04" )
   END_RUNG wire#w1
   RUNG wire#w1
      I_Coil( #TS_EQ01MA02.AutDir1 )
   END_RUNG
   // the same network as SCL:
   #TS_EQ01MA02.AutDir2 := NOT "STATUS_410".DrainMode OR "STATUS_Zone000"."EQ01-BL04";
   #TS_EQ01MA02.AutDir1 := NOT #TS_EQ01MA02.AutDir2;
END_REGION

REGION Network 42: EQ01-MA02 - Valve control
   RUNG wire#powerrail
      #"SF_EQ01-MA02"(IB1ASens := wire#w1, IB1BSens := wire#w2, IS_ZoneM := "STATUS_Zone400".Station410_Mode.Main, IS_ZoneS := "STATUS_Zone400".Station410_Mode.Specific, IB1GenRelDir1 := #TS_EQ01MA02.GenRelDir1, IB1IntlDir1 := #TS_EQ01MA02.IntlDir1, IB1AutDir1 := #TS_EQ01MA02.AutDir1, IB1StartPressDir1 := "STDLog0", IB1ManDir1 := #TS_EQ01MA02.ManDir1, IB1AHold := "STDLog0", IT_ADlyPosTime :=, IT_AMoveErrTime := T#20s, IT_APosErrTime :=, IB1GenRelDir2 := #TS_EQ01MA02.GenRelDir2, IB1IntlDir2 := #TS_EQ01MA02.IntlDir2, IB1AutDir2 := #TS_EQ01MA02.AutDir2, IB1StartPressDir2 := "STDLog0", IB1ManDir2 := #TS_EQ01MA02.ManDir2, IB1BHold := "STDLog0", IT_BDlyPosTime :=, IT_BMoveErrTime := T#20s, IT_BPosErrTime :=, IB1BrkUsed :=, IT_BrkOnTime :=, IT_BrkOffTime :=, IT_Leav := T#2s, IB1AlmSupp := "STATUS_Zone400".Station410_Mode.Specific.AlmSupp, IB1ExtErr :=, XS_Parameter := "HMI_PARAM_410"."EQ01-MA02", XS_Command := "HMI_CMD_410"."EQ01-MA02", OS_Status => "STATUS_410"."EQ01-MA02", OB1OutDir1 => "410UH31-KF01V_A1", OB1OutDir2 => "410UH31-KF01R_A1", OB1BrkRel =>)
   END_RUNG
   RUNG wire#powerrail
      Contact( "STATUS_410"."EQ01-MA02_24" )
      I_Contact( "STATUS_410"."EQ01-MA02_20" )
   END_RUNG wire#w1
   RUNG wire#powerrail
      Contact( "STATUS_410"."EQ01-MA02_20" )
      I_Contact( "STATUS_410"."EQ01-MA02_24" )
   END_RUNG wire#w2
   // the same network as SCL:
   #"SF_EQ01-MA02"(IS_ZoneM := "STATUS_Zone400".Station410_Mode.Main,   // "STD_Valve2WB"
                   IS_ZoneS := "STATUS_Zone400".Station410_Mode.Specific,
                   IB1GenRelDir1 := #TS_EQ01MA02.GenRelDir1,
                   IB1IntlDir1 := #TS_EQ01MA02.IntlDir1,
                   IB1AutDir1 := #TS_EQ01MA02.AutDir1,
                   IB1StartPressDir1 := "STDLog0",
                   IB1ManDir1 := #TS_EQ01MA02.ManDir1,
                   IB1ASens := "STATUS_410"."EQ01-MA02_24" AND NOT "STATUS_410"."EQ01-MA02_20",
                   IB1AHold := "STDLog0",
                   IT_AMoveErrTime := T#20s,
                   IB1GenRelDir2 := #TS_EQ01MA02.GenRelDir2,
                   IB1IntlDir2 := #TS_EQ01MA02.IntlDir2,
                   IB1AutDir2 := #TS_EQ01MA02.AutDir2,
                   IB1StartPressDir2 := "STDLog0",
                   IB1ManDir2 := #TS_EQ01MA02.ManDir2,
                   IB1BSens := "STATUS_410"."EQ01-MA02_20" AND NOT "STATUS_410"."EQ01-MA02_24",
                   IB1BHold := "STDLog0",
                   IT_BMoveErrTime := T#20s,
                   IT_Leav := T#2s,
                   IB1AlmSupp := "STATUS_Zone400".Station410_Mode.Specific.AlmSupp,
                   XS_Parameter := "HMI_PARAM_410"."EQ01-MA02",
                   XS_Command := "HMI_CMD_410"."EQ01-MA02",
                   OS_Status => "STATUS_410"."EQ01-MA02",
                   OB1OutDir1 => "410UH31-KF01V_A1",
                   OB1OutDir2 => "410UH31-KF01R_A1");
END_REGION

REGION Network 43: ********** Circulation Valve EQ01-MA03 **********
END_REGION

REGION Network 44: EQ01-MA03 - General releases
   RUNG wire#powerrail
      Contact( #SB1_PowerOk )
      Coil( #TS_EQ01MA03.GenRelDir1 )
   END_RUNG
   RUNG wire#powerrail
      Contact( #SB1_PowerOk )
      Coil( #TS_EQ01MA03.GenRelDir2 )
   END_RUNG
   // the same network as SCL:
   #TS_EQ01MA03.GenRelDir1 := #SB1_PowerOk;
   #TS_EQ01MA03.GenRelDir2 := #SB1_PowerOk;
END_REGION

REGION Network 45: EQ01-MA03 - Interlocks
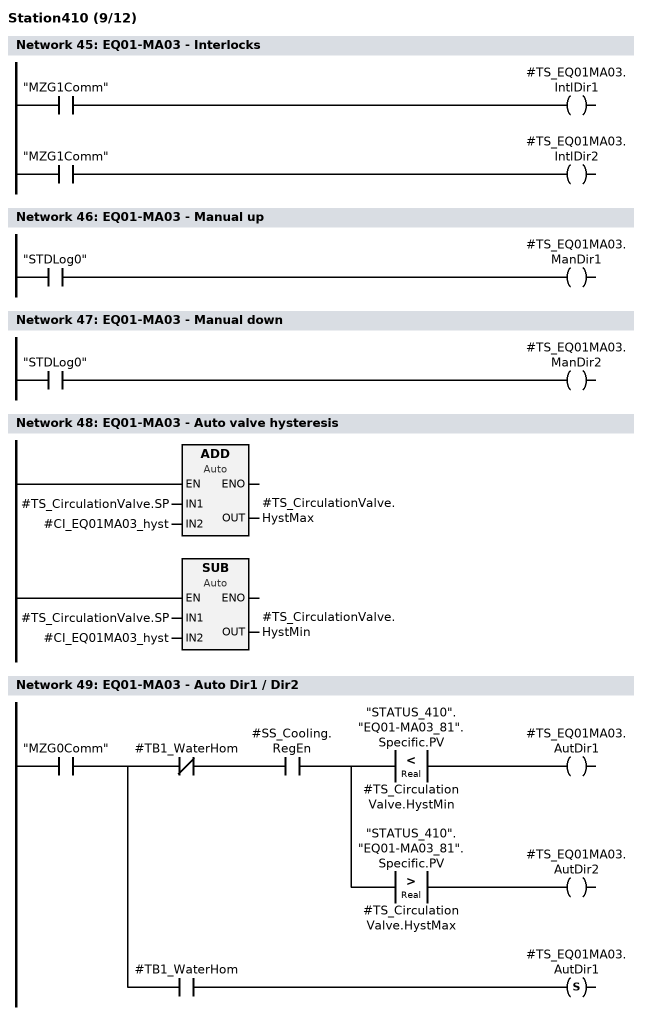
   RUNG wire#powerrail
      Contact( "MZG1Comm" )
      Coil( #TS_EQ01MA03.IntlDir1 )
   END_RUNG
   RUNG wire#powerrail
      Contact( "MZG1Comm" )
      Coil( #TS_EQ01MA03.IntlDir2 )
   END_RUNG
   // the same network as SCL:
   #TS_EQ01MA03.IntlDir1 := "MZG1Comm";
   #TS_EQ01MA03.IntlDir2 := "MZG1Comm";
END_REGION

REGION Network 46: EQ01-MA03 - Manual up
   RUNG wire#powerrail
      Contact( "STDLog0" )
      Coil( #TS_EQ01MA03.ManDir1 )
   END_RUNG
   // the same network as SCL:
   #TS_EQ01MA03.ManDir1 := "STDLog0";
END_REGION

REGION Network 47: EQ01-MA03 - Manual down
   RUNG wire#powerrail
      Contact( "STDLog0" )
      Coil( #TS_EQ01MA03.ManDir2 )
   END_RUNG
   // the same network as SCL:
   #TS_EQ01MA03.ManDir2 := "STDLog0";
END_REGION

REGION Network 48: EQ01-MA03 - Auto valve hysteresis
   RUNG wire#powerrail
      Add(in1 := #TS_CirculationValve.SP, in2 := #CI_EQ01MA03_hyst, out => #TS_CirculationValve.HystMax)
   END_RUNG
   RUNG wire#powerrail
      Sub(in1 := #TS_CirculationValve.SP, in2 := #CI_EQ01MA03_hyst, out => #TS_CirculationValve.HystMin)
   END_RUNG
   // the same network as SCL:
   #TS_CirculationValve.HystMax := #TS_CirculationValve.SP + #CI_EQ01MA03_hyst;
   #TS_CirculationValve.HystMin := #TS_CirculationValve.SP - #CI_EQ01MA03_hyst;
END_REGION

REGION Network 49: EQ01-MA03 - Auto Dir1 / Dir2
   RUNG wire#powerrail
      Contact( "MZG0Comm" )
      wire#w1
      I_Contact( #TB1_WaterHom )
      Contact( #SS_Cooling.RegEn )
      wire#w2
      { S7_Templates := "SrcType := Real" } LT_Contact(in1 := "STATUS_410"."EQ01-MA03_81".Specific.PV, in2 := #TS_CirculationValve.HystMin)
      Coil( #TS_EQ01MA03.AutDir1 )
   END_RUNG
   RUNG wire#w2
      { S7_Templates := "SrcType := Real" } GT_Contact(in1 := "STATUS_410"."EQ01-MA03_81".Specific.PV, in2 := #TS_CirculationValve.HystMax)
      Coil( #TS_EQ01MA03.AutDir2 )
   END_RUNG
   RUNG wire#w1
      Contact( #TB1_WaterHom )
      S_Coil( #TS_EQ01MA03.AutDir1 )
   END_RUNG
   // the same network as SCL:
   #_w1 := "MZG0Comm" AND NOT #TB1_WaterHom AND #SS_Cooling.RegEn;
   #TS_EQ01MA03.AutDir1 := #_w1 AND ("STATUS_410"."EQ01-MA03_81".Specific.PV < #TS_CirculationValve.HystMin);
   #TS_EQ01MA03.AutDir2 := #_w1 AND ("STATUS_410"."EQ01-MA03_81".Specific.PV > #TS_CirculationValve.HystMax);
   IF "MZG0Comm" AND #TB1_WaterHom THEN #TS_EQ01MA03.AutDir1 := TRUE; END_IF;
END_REGION

REGION Network 50: EQ01-MA03 - Valve control
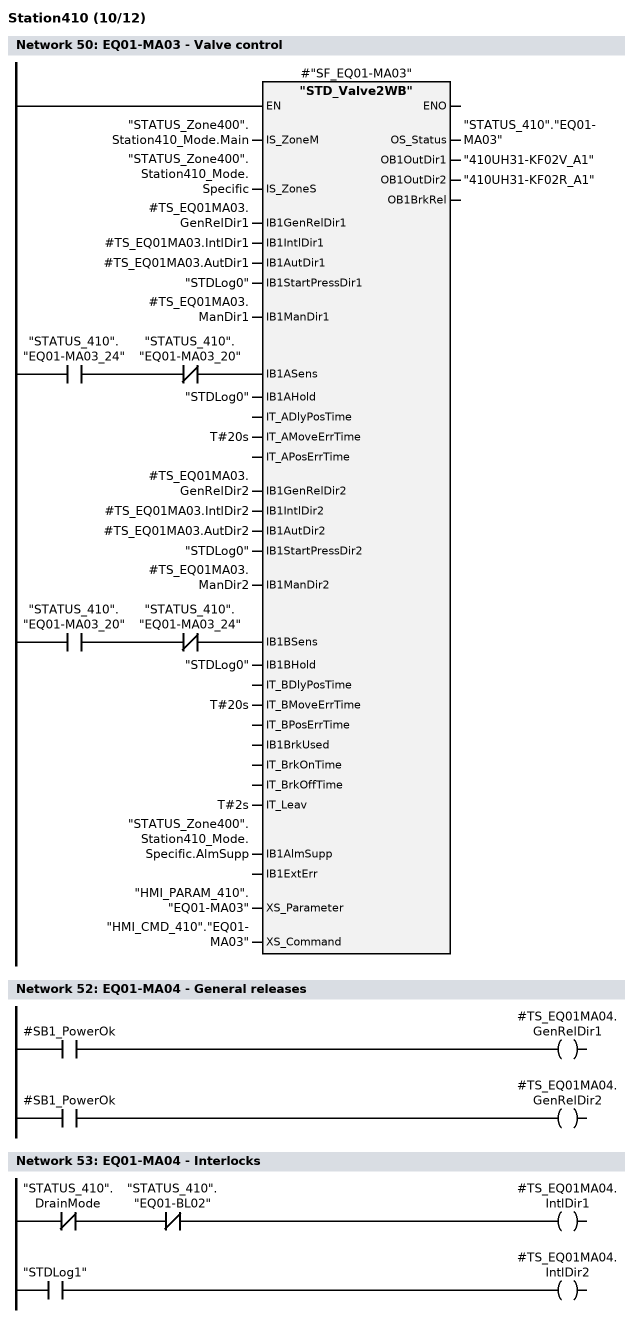
   RUNG wire#powerrail
      #"SF_EQ01-MA03"(IB1ASens := wire#w1, IB1BSens := wire#w2, IS_ZoneM := "STATUS_Zone400".Station410_Mode.Main, IS_ZoneS := "STATUS_Zone400".Station410_Mode.Specific, IB1GenRelDir1 := #TS_EQ01MA03.GenRelDir1, IB1IntlDir1 := #TS_EQ01MA03.IntlDir1, IB1AutDir1 := #TS_EQ01MA03.AutDir1, IB1StartPressDir1 := "STDLog0", IB1ManDir1 := #TS_EQ01MA03.ManDir1, IB1AHold := "STDLog0", IT_ADlyPosTime :=, IT_AMoveErrTime := T#20s, IT_APosErrTime :=, IB1GenRelDir2 := #TS_EQ01MA03.GenRelDir2, IB1IntlDir2 := #TS_EQ01MA03.IntlDir2, IB1AutDir2 := #TS_EQ01MA03.AutDir2, IB1StartPressDir2 := "STDLog0", IB1ManDir2 := #TS_EQ01MA03.ManDir2, IB1BHold := "STDLog0", IT_BDlyPosTime :=, IT_BMoveErrTime := T#20s, IT_BPosErrTime :=, IB1BrkUsed :=, IT_BrkOnTime :=, IT_BrkOffTime :=, IT_Leav := T#2s, IB1AlmSupp := "STATUS_Zone400".Station410_Mode.Specific.AlmSupp, IB1ExtErr :=, XS_Parameter := "HMI_PARAM_410"."EQ01-MA03", XS_Command := "HMI_CMD_410"."EQ01-MA03", OS_Status => "STATUS_410"."EQ01-MA03", OB1OutDir1 => "410UH31-KF02V_A1", OB1OutDir2 => "410UH31-KF02R_A1", OB1BrkRel =>)
   END_RUNG
   RUNG wire#powerrail
      Contact( "STATUS_410"."EQ01-MA03_24" )
      I_Contact( "STATUS_410"."EQ01-MA03_20" )
   END_RUNG wire#w1
   RUNG wire#powerrail
      Contact( "STATUS_410"."EQ01-MA03_20" )
      I_Contact( "STATUS_410"."EQ01-MA03_24" )
   END_RUNG wire#w2
   // the same network as SCL:
   #"SF_EQ01-MA03"(IS_ZoneM := "STATUS_Zone400".Station410_Mode.Main,   // "STD_Valve2WB"
                   IS_ZoneS := "STATUS_Zone400".Station410_Mode.Specific,
                   IB1GenRelDir1 := #TS_EQ01MA03.GenRelDir1,
                   IB1IntlDir1 := #TS_EQ01MA03.IntlDir1,
                   IB1AutDir1 := #TS_EQ01MA03.AutDir1,
                   IB1StartPressDir1 := "STDLog0",
                   IB1ManDir1 := #TS_EQ01MA03.ManDir1,
                   IB1ASens := "STATUS_410"."EQ01-MA03_24" AND NOT "STATUS_410"."EQ01-MA03_20",
                   IB1AHold := "STDLog0",
                   IT_AMoveErrTime := T#20s,
                   IB1GenRelDir2 := #TS_EQ01MA03.GenRelDir2,
                   IB1IntlDir2 := #TS_EQ01MA03.IntlDir2,
                   IB1AutDir2 := #TS_EQ01MA03.AutDir2,
                   IB1StartPressDir2 := "STDLog0",
                   IB1ManDir2 := #TS_EQ01MA03.ManDir2,
                   IB1BSens := "STATUS_410"."EQ01-MA03_20" AND NOT "STATUS_410"."EQ01-MA03_24",
                   IB1BHold := "STDLog0",
                   IT_BMoveErrTime := T#20s,
                   IT_Leav := T#2s,
                   IB1AlmSupp := "STATUS_Zone400".Station410_Mode.Specific.AlmSupp,
                   XS_Parameter := "HMI_PARAM_410"."EQ01-MA03",
                   XS_Command := "HMI_CMD_410"."EQ01-MA03",
                   OS_Status => "STATUS_410"."EQ01-MA03",
                   OB1OutDir1 => "410UH31-KF02V_A1",
                   OB1OutDir2 => "410UH31-KF02R_A1");
END_REGION

REGION Network 51: ********** Filling Valve EQ01-MA04 **********
END_REGION

REGION Network 52: EQ01-MA04 - General releases
   RUNG wire#powerrail
      Contact( #SB1_PowerOk )
      Coil( #TS_EQ01MA04.GenRelDir1 )
   END_RUNG
   RUNG wire#powerrail
      Contact( #SB1_PowerOk )
      Coil( #TS_EQ01MA04.GenRelDir2 )
   END_RUNG
   // the same network as SCL:
   #TS_EQ01MA04.GenRelDir1 := #SB1_PowerOk;
   #TS_EQ01MA04.GenRelDir2 := #SB1_PowerOk;
END_REGION

REGION Network 53: EQ01-MA04 - Interlocks
   RUNG wire#powerrail
      I_Contact( "STATUS_410".DrainMode )
      I_Contact( "STATUS_410"."EQ01-BL02" )
      Coil( #TS_EQ01MA04.IntlDir1 )
   END_RUNG
   RUNG wire#powerrail
      Contact( "STDLog1" )
      Coil( #TS_EQ01MA04.IntlDir2 )
   END_RUNG
   // the same network as SCL:
   #TS_EQ01MA04.IntlDir1 := NOT "STATUS_410".DrainMode AND NOT "STATUS_410"."EQ01-BL02";
   #TS_EQ01MA04.IntlDir2 := "STDLog1";
END_REGION

REGION Network 54: EQ01-MA04 - Manual up
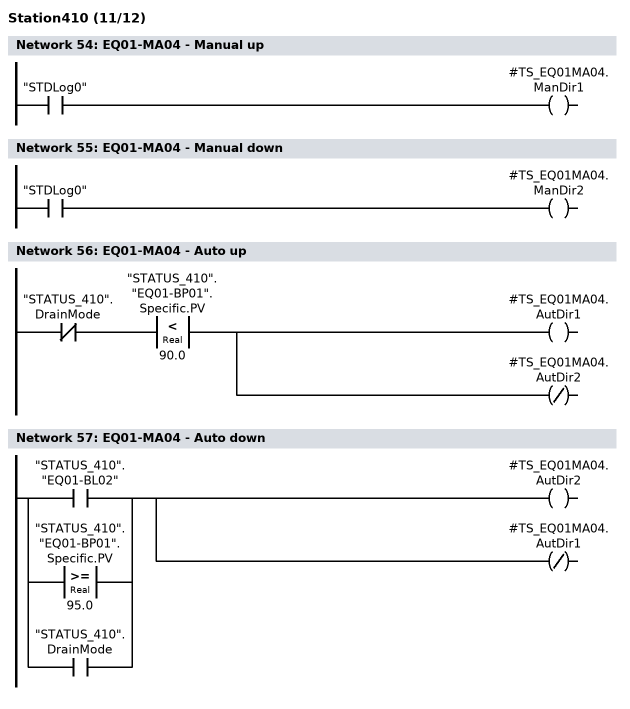
   RUNG wire#powerrail
      Contact( "STDLog0" )
      Coil( #TS_EQ01MA04.ManDir1 )
   END_RUNG
   // the same network as SCL:
   #TS_EQ01MA04.ManDir1 := "STDLog0";
END_REGION

REGION Network 55: EQ01-MA04 - Manual down
   RUNG wire#powerrail
      Contact( "STDLog0" )
      Coil( #TS_EQ01MA04.ManDir2 )
   END_RUNG
   // the same network as SCL:
   #TS_EQ01MA04.ManDir2 := "STDLog0";
END_REGION

REGION Network 56: EQ01-MA04 - Auto up
   RUNG wire#powerrail
      I_Contact( "STATUS_410".DrainMode )
      { S7_Templates := "SrcType := Real" } LT_Contact(in1 := "STATUS_410"."EQ01-BP01".Specific.PV, in2 := 90.0)
      wire#w1
      Coil( #TS_EQ01MA04.AutDir1 )
   END_RUNG
   RUNG wire#w1
      I_Coil( #TS_EQ01MA04.AutDir2 )
   END_RUNG
   // the same network as SCL:
   #TS_EQ01MA04.AutDir1 := NOT "STATUS_410".DrainMode AND ("STATUS_410"."EQ01-BP01".Specific.PV < 90.0);
   #TS_EQ01MA04.AutDir2 := NOT #TS_EQ01MA04.AutDir1;
END_REGION

REGION Network 57: EQ01-MA04 - Auto down
   RUNG wire#powerrail
      Contact( "STATUS_410"."EQ01-BL02" )
      wire#w1
      Coil( #TS_EQ01MA04.AutDir2 )
   END_RUNG
   RUNG wire#powerrail
      { S7_Templates := "SrcType := Real" } GE_Contact(in1 := "STATUS_410"."EQ01-BP01".Specific.PV, in2 := 95.0)
   END_RUNG wire#w1
   RUNG wire#powerrail
      Contact( "STATUS_410".DrainMode )
   END_RUNG wire#w1
   RUNG wire#w1
      I_Coil( #TS_EQ01MA04.AutDir1 )
   END_RUNG
   // the same network as SCL:
   #TS_EQ01MA04.AutDir2 := "STATUS_410"."EQ01-BL02" OR ("STATUS_410"."EQ01-BP01".Specific.PV >= 95.0) OR "STATUS_410".DrainMode;
   #TS_EQ01MA04.AutDir1 := NOT #TS_EQ01MA04.AutDir2;
END_REGION

REGION Network 58: EQ01-MA04 - Valve control
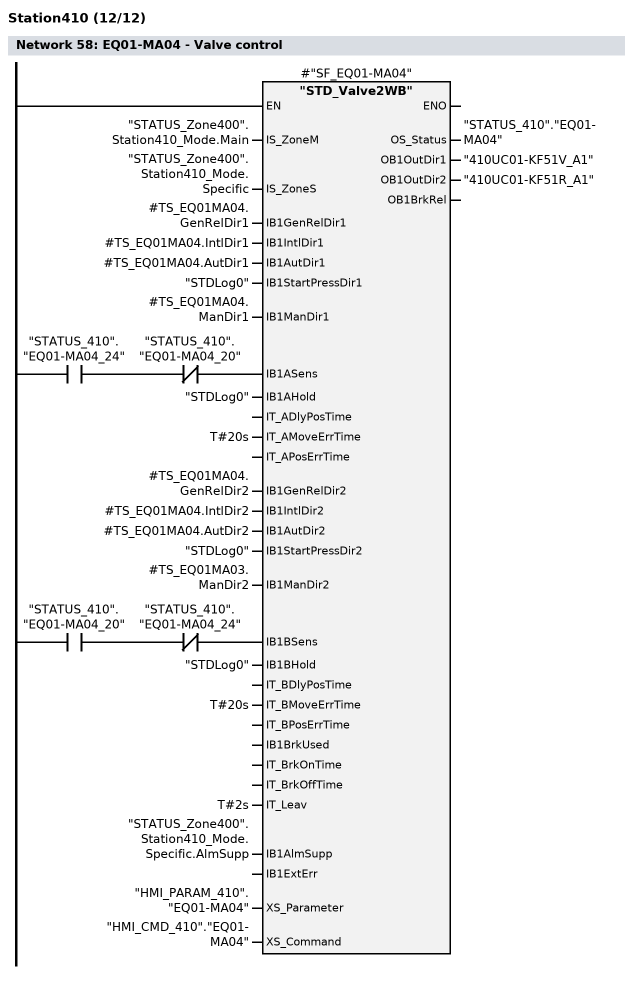
   RUNG wire#powerrail
      #"SF_EQ01-MA04"(IB1ASens := wire#w1, IB1BSens := wire#w2, IS_ZoneM := "STATUS_Zone400".Station410_Mode.Main, IS_ZoneS := "STATUS_Zone400".Station410_Mode.Specific, IB1GenRelDir1 := #TS_EQ01MA04.GenRelDir1, IB1IntlDir1 := #TS_EQ01MA04.IntlDir1, IB1AutDir1 := #TS_EQ01MA04.AutDir1, IB1StartPressDir1 := "STDLog0", IB1ManDir1 := #TS_EQ01MA04.ManDir1, IB1AHold := "STDLog0", IT_ADlyPosTime :=, IT_AMoveErrTime := T#20s, IT_APosErrTime :=, IB1GenRelDir2 := #TS_EQ01MA04.GenRelDir2, IB1IntlDir2 := #TS_EQ01MA04.IntlDir2, IB1AutDir2 := #TS_EQ01MA04.AutDir2, IB1StartPressDir2 := "STDLog0", IB1ManDir2 := #TS_EQ01MA03.ManDir2, IB1BHold := "STDLog0", IT_BDlyPosTime :=, IT_BMoveErrTime := T#20s, IT_BPosErrTime :=, IB1BrkUsed :=, IT_BrkOnTime :=, IT_BrkOffTime :=, IT_Leav := T#2s, IB1AlmSupp := "STATUS_Zone400".Station410_Mode.Specific.AlmSupp, IB1ExtErr :=, XS_Parameter := "HMI_PARAM_410"."EQ01-MA04", XS_Command := "HMI_CMD_410"."EQ01-MA04", OS_Status => "STATUS_410"."EQ01-MA04", OB1OutDir1 => "410UC01-KF51V_A1", OB1OutDir2 => "410UC01-KF51R_A1", OB1BrkRel =>)
   END_RUNG
   RUNG wire#powerrail
      Contact( "STATUS_410"."EQ01-MA04_24" )
      I_Contact( "STATUS_410"."EQ01-MA04_20" )
   END_RUNG wire#w1
   RUNG wire#powerrail
      Contact( "STATUS_410"."EQ01-MA04_20" )
      I_Contact( "STATUS_410"."EQ01-MA04_24" )
   END_RUNG wire#w2
   // the same network as SCL:
   #"SF_EQ01-MA04"(IS_ZoneM := "STATUS_Zone400".Station410_Mode.Main,   // "STD_Valve2WB"
                   IS_ZoneS := "STATUS_Zone400".Station410_Mode.Specific,
                   IB1GenRelDir1 := #TS_EQ01MA04.GenRelDir1,
                   IB1IntlDir1 := #TS_EQ01MA04.IntlDir1,
                   IB1AutDir1 := #TS_EQ01MA04.AutDir1,
                   IB1StartPressDir1 := "STDLog0",
                   IB1ManDir1 := #TS_EQ01MA04.ManDir1,
                   IB1ASens := "STATUS_410"."EQ01-MA04_24" AND NOT "STATUS_410"."EQ01-MA04_20",
                   IB1AHold := "STDLog0",
                   IT_AMoveErrTime := T#20s,
                   IB1GenRelDir2 := #TS_EQ01MA04.GenRelDir2,
                   IB1IntlDir2 := #TS_EQ01MA04.IntlDir2,
                   IB1AutDir2 := #TS_EQ01MA04.AutDir2,
                   IB1StartPressDir2 := "STDLog0",
                   IB1ManDir2 := #TS_EQ01MA03.ManDir2,
                   IB1BSens := "STATUS_410"."EQ01-MA04_20" AND NOT "STATUS_410"."EQ01-MA04_24",
                   IB1BHold := "STDLog0",
                   IT_BMoveErrTime := T#20s,
                   IT_Leav := T#2s,
                   IB1AlmSupp := "STATUS_Zone400".Station410_Mode.Specific.AlmSupp,
                   XS_Parameter := "HMI_PARAM_410"."EQ01-MA04",
                   XS_Command := "HMI_CMD_410"."EQ01-MA04",
                   OS_Status => "STATUS_410"."EQ01-MA04",
                   OB1OutDir1 => "410UC01-KF51V_A1",
                   OB1OutDir2 => "410UC01-KF51R_A1");
END_REGION
END_FUNCTION_BLOCK
